{attribute addProperty BoxType "AX8108-0000-0041-0041"}
{attribute addProperty Id "Ch_A_Velocity_sensor_actual_value_invalidAT %I*BOOL811Ch_A_Position_actual_value_invalidAT %I*BOOL812Ch_A_1st_Additional_position_actual_value_invalidAT %I*BOOL813Ch_A_2nd_Additional_position_actual_value_invalidAT %I*BOOL814Ch_A_StatuswordAT %I*UINT1620Ch_A_Position_actual_valueAT %I*DINT3240Ch_A_Velocity_actual_valueAT %I*DINT3240"}
{attribute addProperty CRC "1519847663"}
{attribute addProperty SizeInBites "112"}
{attribute addProperty SizeInBytes "14"}
TYPE Ch_A_AxisMain_Inputs_5A9708EF :
STRUCT
	{attribute addProperty Name "Ch_A_Velocity_sensor_actual_value_invalid"}
	Ch_A_Velocity_sensor_actual_value_invalid AT %I* : BOOL;
	{attribute addProperty Name "Ch_A_Position_actual_value_invalid"}
	Ch_A_Position_actual_value_invalid AT %I* : BOOL;
	{attribute addProperty Name "Ch_A_1st_Additional_position_actual_value_invalid"}
	Ch_A_1st_Additional_position_actual_value_invalid AT %I* : BOOL;
	{attribute addProperty Name "Ch_A_2nd_Additional_position_actual_value_invalid"}
	Ch_A_2nd_Additional_position_actual_value_invalid AT %I* : BOOL;
	{attribute addProperty Name "Ch_A_Statusword"}
	Ch_A_Statusword AT %I* : UINT;
	{attribute addProperty Name "Ch_A_Position_actual_value"}
	Ch_A_Position_actual_value AT %I* : DINT;
	{attribute addProperty Name "Ch_A_Velocity_actual_value"}
	Ch_A_Velocity_actual_value AT %I* : DINT;
END_STRUCT
END_TYPE

(* stored: Version 1.2.0.0, ProductVersion 3.1.4024.9
   DUT Ch_A_AxisMain_Inputs_5A9708EF: Id {54374a2c-e495-4caa-b4b9-5d859047772b} *)
